FUNCTION_BLOCK FB_EstacionFinalizar_SFC
VAR_INPUT
    // SFC-Flags
    SFCPause: BOOL;
    SFCReset: BOOL;
    
    // Indicadores de sincronizacion
    Ack: BOOL := TRUE;
    Execute: BOOL;
    
    // Parametros
    TpoFinalizacion: TIME := T#1S;
END_VAR
VAR_OUTPUT
    // Indicadores de sincronizacion
    Done: BOOL;
    Ready: BOOL;
END_VAR
VAR
END_VAR

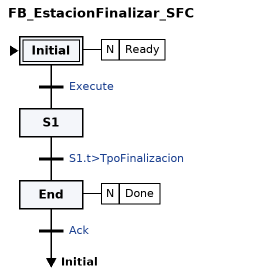
INITIAL_STEP Initial:
    Ready(N);
END_STEP
TRANSITION FROM Initial TO S1
    := Execute;
END_TRANSITION
STEP S1:
END_STEP
TRANSITION FROM S1 TO End
    := S1.t>TpoFinalizacion;
END_TRANSITION
STEP End:
    Done(N);
END_STEP
TRANSITION FROM End TO Initial
    := Ack;
END_TRANSITION

END_FUNCTION_BLOCK

(* stored: Version 1.1.0.1, ProductVersion 3.1.4024.12
   POU FB_EstacionFinalizar_SFC: Id {4f954952-ece8-4689-b1b8-f2e82ec4d38c}, SpecialFunc None *)
